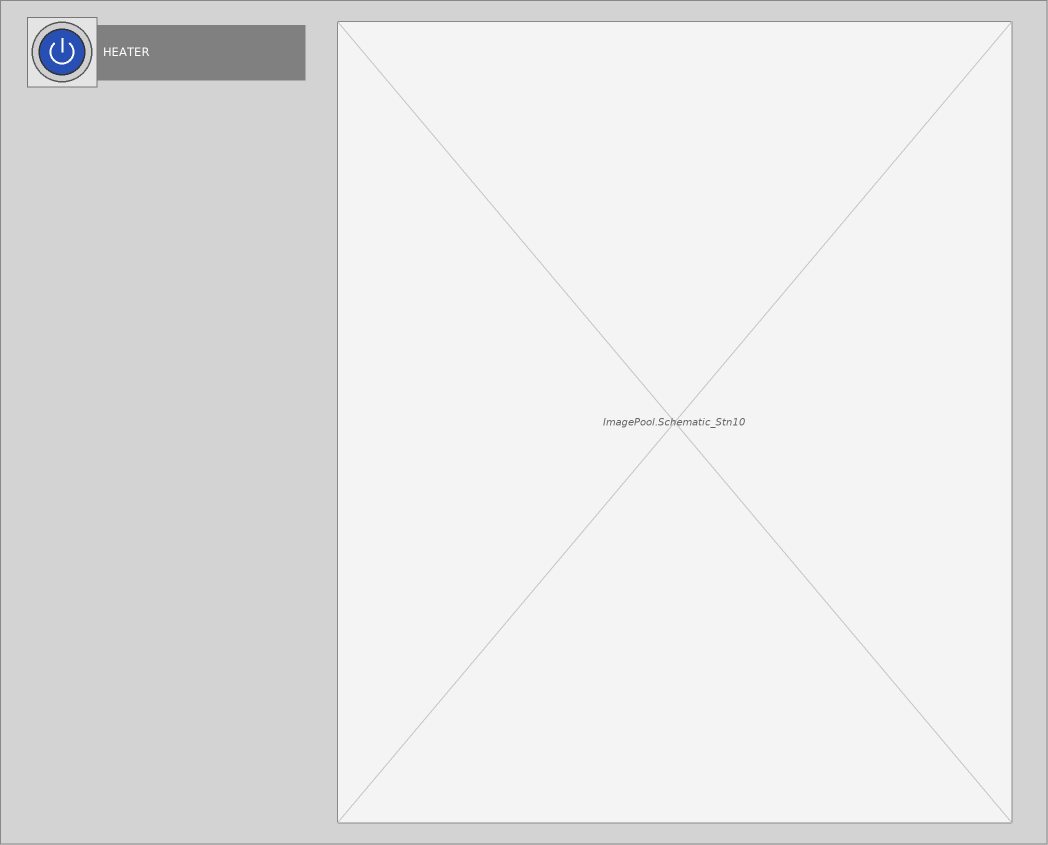
VISUALIZATION Recipe_Station10  // 1048x845
    Rectangle (0,0 1048x845)
    Label (100,44 163x16)
    RoundedRectangle (74,25 231x55)
    Label (100,44 151x16), "HEATER"
    PowerSwitch (27,17 70x70), variable: DSScrMapSSUR.DsSubRecipeMemory.bOut2EnProTankHeater, behaviour: TOGGLE, style: Switch-PowerSwitch-Blue
    Image (337,21 675x802), image: ImagePool.Schematic_Stn10
END_VISUALIZATION

(* stored: Version 1.1.0.1, ProductVersion 3.1.4024.12
   Visu Recipe_Station10: Id {ef019a8b-d359-4faf-96aa-922ae382e385} *)
